(* PLC project Unnamed, Unknown Unnamed 1 *)
(* stored: creationDateTime 2026-04-06T14:45:05, modificationDateTime 2026-04-06T14:45:05 *)

FUNCTION_BLOCK Wifi_Scanner
  VAR
    hasBeenInitialized : BOOL := 0;
  END_VAR

            {{
WIFI_SCANNER_VARS vars;
}}
if hasBeenInitialized = False then
{{
wifi_scanner_setup(&vars);
}}
hasBeenInitialized := True;
end_if;
{{
wifi_scanner_loop(&vars);
}}
          
END_FUNCTION_BLOCK

PROGRAM main
  VAR
    LED_out AT %QX0.0 : BOOL;
  END_VAR
  VAR
    Waktu_Blink : TIME := T#1s;
    Timer1 : TON;
    Timer2 : TON;
    WIFI_SCANNER1 : Wifi_Scanner;
  END_VAR

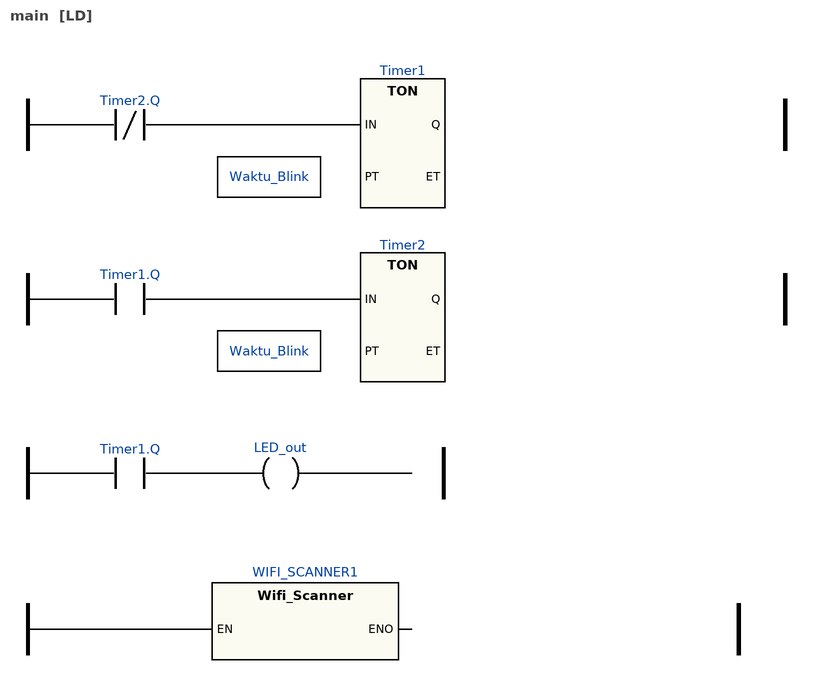
(* LD diagram, written out as Structured Text *)
LED_out := Timer1.Q;
Timer1(IN := NOT Timer2.Q, PT := Waktu_Blink);
Timer2(IN := Timer1.Q, PT := Waktu_Blink);
WIFI_SCANNER1();
END_PROGRAM

CONFIGURATION Config0
  RESOURCE Res0 ON PLC
    TASK task0(INTERVAL := T#20ms, PRIORITY := 1);
    PROGRAM instance0 WITH task0 : main;
  END_RESOURCE
END_CONFIGURATION
